FUNCTION F_FormatStringEx4 : T_MaxString
VAR_INPUT
	Format	: T_MaxString;
	arg1	: T_MaxString;
	arg2	: T_MaxString;
	arg3	: T_MaxString;
	arg4	: T_MaxString;
END_VAR
VAR
    FB_FormatString1 : FB_FormatString;
END_VAR



FB_FormatString1(
	sFormat:= Format, 
	arg1:= F_STRING(arg1), 
	arg2:= F_STRING(arg2),
	arg3:= F_STRING(arg3), 
	arg4:= F_STRING(arg4), 
	arg5:= , 
	arg6:= , 
	arg7:= , 
	arg8:= , 
	arg9:= , 
	arg10:= , 
	bError=> , 
	nErrId=> , 
	sOut=> F_FormatStringEx4);

END_FUNCTION

(* stored: Version 1.1.0.1, ProductVersion 3.1.4024.3
   POU F_FormatStringEx4: Id {1eaf65ad-ac62-0dd9-316c-49dde2887e49}, SpecialFunc None *)
